(* IEC 61131-3 sources: twincat-conveyor-simulator/TwinCAT/PLC/GVLs, 3 files *)

(* ---- GVL_HMI_Engineering.st ---- *)
{attribute 'qualified_only'}
VAR_GLOBAL
    bAutoSimulationEnabled : BOOL := TRUE;
    bManualEntrySensor     : BOOL := FALSE;
    bManualExitSensor      : BOOL := FALSE;
    bInjectFault           : BOOL := FALSE;
    bResetCounter          : BOOL := FALSE;

    bSimulatedEntrySensor  : BOOL := FALSE;
    bSimulatedExitSensor   : BOOL := FALSE;
    nSimulationStep        : UINT := 0;
END_VAR

(* ---- GVL_HMI_Operator.st ---- *)
{attribute 'qualified_only'}
VAR_GLOBAL
    bStartCommand  : BOOL := FALSE;
    bStopCommand   : BOOL := FALSE;
    bResetCommand  : BOOL := FALSE;
    bEmergencyStop : BOOL := FALSE;
    stStatus       : ST_ConveyorStatus;
END_VAR

(* ---- GVL_IO.st ---- *)
{attribute 'qualified_only'}
VAR_GLOBAL
    bEntrySensorInput    : BOOL := FALSE;
    bExitSensorInput     : BOOL := FALSE;
    bConveyorMotorOutput : BOOL := FALSE;
END_VAR
